// TIA Portal V20 export
TYPE "UDT_RunTime_Steuern"
   STRUCT
      run_Time : Struct
         seconds : Int;
         minutes : Int;
         hours : Real;
         days : Real;
         years : Real;
      END_STRUCT;
   END_STRUCT;
END_TYPE
